PROGRAM PRG_ProcessCellSimulation

fbMachine.Update();

END_PROGRAM

(* stored: Version 1.1.0.1, ProductVersion 3.1.4024.12
   POU PRG_ProcessCellSimulation: Id {c2a13f8d-2794-4486-b5dd-3ad3830b6f94}, SpecialFunc None *)
